// TIA Portal V18 export
VAR_GLOBAL   // PLC tag table "STEP7 classic symbols"
   "ClockMemory0.8s" AT %M0.4 : Bool;
   "ClockMemory0.5s" AT %M0.3 : Bool;
   "ClockMemory0.4s" AT %M0.2 : Bool;
   "ClockMemory0.2s" AT %M0.1 : Bool;
   "ClockMemory0.1s" AT %M0.0 : Bool;
   ClockMemory2s AT %M0.7 : Bool;
   "ClockMemory1.6s" AT %M0.6 : Bool;
   ClockMemory1s AT %M0.5 : Bool;
END_VAR
